(* CODESYS project mathlibrary_plc.library
   Company: ITT_MathLibrary
   Description: MathLibrary contains Addition, Division, Multiplication, Square, Subtract, Cube
   Version: 1.0.0
   Placeholder: MathLibrary
   Author: Krishnpal
   Title: MathLibrary

Project tree, tasks and I/O mapping:
  libraries: Tc2_Standard, * (Beckhoff Automation GmbH); Tc2_System, * (Beckhoff Automation GmbH); Tc3_Module, * (Beckhoff Automation GmbH)
  POUs/
    function block FB_Addition [ST]
    function block FB_Division [ST]
    function block FB_Multiplication [ST]
    function block FB_Square [ST]
    function block FB_Subtract [ST]
    program MAIN [ST]
  Version/
    global variables Global_Version
  function block FB_Cube [ST]
*)

// Version/Global_Version
{attribute 'TcGenerated'}
{attribute 'no-analysis'}
{attribute 'linkalways'}
// This function has been automatically generated from the project information.
VAR_GLOBAL CONSTANT
	{attribute 'const_non_replaced'}
	stLibVersion_MathLibrary : ST_LibVersion := (iMajor := 1, iMinor := 0, iBuild := 0, iRevision := 0, nFlags := 0, sVersion := '1.0.0');
END_VAR

// POUs/FB_Addition
FUNCTION_BLOCK FB_Addition
VAR_INPUT
	iNum1 : INT;
	iNum2 : INT;
END_VAR
VAR_OUTPUT
	iResult : INT;
END_VAR

iResult := iNum1 + iNum2;

END_FUNCTION_BLOCK

// POUs/FB_Division
FUNCTION_BLOCK FB_Division
VAR_INPUT
	iNum1 : INT;
	iNum2 : INT;
END_VAR
VAR_OUTPUT
	iResult : REAL;
	statusMessage : STRING(30);
END_VAR

IF iNum2 > 0 THEN
	iResult := iNum1/iNum2;
ELSE
	statusMessage := 'Value should be greater than 0';
END_IF

END_FUNCTION_BLOCK

// POUs/FB_Multiplication
FUNCTION_BLOCK FB_Multiplication
VAR_INPUT
	iVar1 : INT;
	iVar2 : INT;
END_VAR
VAR_OUTPUT
	iResult : INT;
END_VAR

iResult := iVar1 * iVar2;

END_FUNCTION_BLOCK

// POUs/FB_Square
FUNCTION_BLOCK FB_Square
VAR_INPUT
	iNum : INT;
END_VAR
VAR_OUTPUT
	iResult : INT;
END_VAR

iResult := iNum * iNum;

END_FUNCTION_BLOCK

// POUs/FB_Subtract
FUNCTION_BLOCK FB_Subtract
VAR_INPUT
	iVar1 : INT;
	iVar2 : INT;
END_VAR
VAR_OUTPUT
	iResult : INT;
END_VAR

iResult := iVar1 - iVar2;

END_FUNCTION_BLOCK

// POUs/MAIN
PROGRAM MAIN
VAR
	fbAddition : FB_Addition;
	fbCube : FB_Cube;
	fbDivision : FB_Division;
	fbMultiplication : FB_Multiplication;
	fbSquare : FB_Square;
	fbSubtract : FB_Subtract;
END_VAR

fbAddition(iNum1:=4, iNum2:=5);
fbCube(iNum := 6);
fbDivision(iNum1:=6,iNum2:=0);
fbMultiplication(iVar1:=8, iVar2:=2);
fbSquare(iNum :=4);
fbSubtract(iVar1:=8, iVar2:=3);

END_PROGRAM

// FB_Cube
FUNCTION_BLOCK FB_Cube
VAR_INPUT
	iNum : INT;
END_VAR
VAR_OUTPUT
	iResult : INT;
END_VAR

iResult := iNum * iNum * iNum ;

END_FUNCTION_BLOCK
